// TIA Portal V19 export
TYPE "ValveMonitor_UDT"
   STRUCT
      Activation : Struct
         ActivationCounter : DInt;
         StrokeDuration : Struct
            Average : Int;   // Average of n1 - n10 Durations in mSec
            count : Int;   // Duration count
            Archive : Struct
               n1 : Int;   // Current Activation Duration
               n2 : Int;   // Previous Activation Duration
               n3 : Int;
               n4 : Int;
               n5 : Int;
               n6 : Int;
               n7 : Int;
               n8 : Int;
               n9 : Int;
               n10 : Int;
            END_STRUCT;
         END_STRUCT;
      END_STRUCT;
      De_Activation : Struct
         De_ActivationCounter : DInt;
         StrokeDuration : Struct
            Average : Int;   // Average of n1 - n10 Durations in mSec
            count : Int;   // Duration count
            Archive : Struct
               n1 : Int;   // Current Activation Duration
               n2 : Int;   // Previous Activation Duration
               n3 : Int;
               n4 : Int;
               n5 : Int;
               n6 : Int;
               n7 : Int;
               n8 : Int;
               n9 : Int;
               n10 : Int;
            END_STRUCT;
         END_STRUCT;
      END_STRUCT;
   END_STRUCT;
END_TYPE
